TYPE E_WashMode :
(
	MODE_Undefiend,
	MODE_WashOutside,
	MODE_WashInside,
	MODE_WashInOutside,
	MODE_DryInside,
	MODE_DryOutside
) USINT;
END_TYPE

(* stored: Version 1.1.0.1, ProductVersion 3.1.4022.10
   DUT E_WashMode: Id {63b07b8f-7178-4dc1-a374-e27b05f3a625} *)
